FUNCTION_BLOCK TcMessage_Ext IMPLEMENTS ITcMessage_Ext
VAR_INPUT
END_VAR
VAR_OUTPUT
END_VAR
VAR
    fbMsg : FB_TcMessage; 
	fbTest : Tc3_EventLogger.FB_TcEvent;
	fbInfo : Tc3_EventLogger.FB_TcSourceInfo;
	_loggerLevel : TcEventSeverity := TcEventSeverity.Info;
END_VAR

PROPERTY PUBLIC LoggerLevel : TcEventSeverity
GET
LoggerLevel := _loggerLevel;
END_GET
SET
_loggerLevel := LoggerLevel;
END_SET
END_PROPERTY

METHOD PUBLIC Send : BOOL
VAR_INPUT
	eventType : Tc3_EventLogger.TcEventEntry;
	args : STRING(255);
END_VAR
IF eventType.eSeverity >= LoggerLevel THEN
	THIS^.fbMsg.CreateEx(eventType, 0);
	THIS^.fbMsg.ipArguments.AddString(args);
	THIS^.fbMsg.Send(0);
	THIS^.fbMsg.Release();
END_IF
END_METHOD

END_FUNCTION_BLOCK

(* stored: Version 1.1.0.1, ProductVersion 3.1.4024.11
   POU TcMessage_Ext: Id {2ca986e9-916e-4607-8394-ce75009d3f97}, SpecialFunc None
   Property LoggerLevel: Id {0fc0c4e3-2c92-463c-817e-81d49d6290e6}
   Get Get: Id {692c3257-9442-4607-8aef-3d73b2262680}
   Set Set: Id {8bbd2b78-98bd-442c-835b-e07b897d2146}
   Method Send: Id {1099518a-0ae3-456e-89fa-82efcf67d371} *)
